// TIA Portal V21 export
FUNCTION_BLOCK "FB101"   // FB101, LAD
TITLE = FB101
{ S7_Optimized_Access := 'TRUE' }
AUTHOR : PRECISE
FAMILY : PRECISE
// TIMER (RETENTIVE)
// stored: AutoNumber false, MemoryReserve 100, SetENOAutomatically false
   VAR_INPUT
      Enable : Bool;
      Running : Bool;
      Reset : Bool;
      SecPulse : Bool;
      AlwaysTrue : Bool;
      TimeBaseSel : Bool;   // Time Base Selection: 0-second/1-minute
      TimeMin : Int;
      TimeSec : Int;
   END_VAR
   VAR_OUTPUT
      Done : Bool;
      TimeMinPV : DInt;
      TimeSecPV : DInt;
   END_VAR
   VAR_IN_OUT
      TimeSV : DInt;
      TimePV : DInt;
      TempBit : Bool;
   END_VAR
BEGIN

REGION Network 1: Set Time Min/Sec
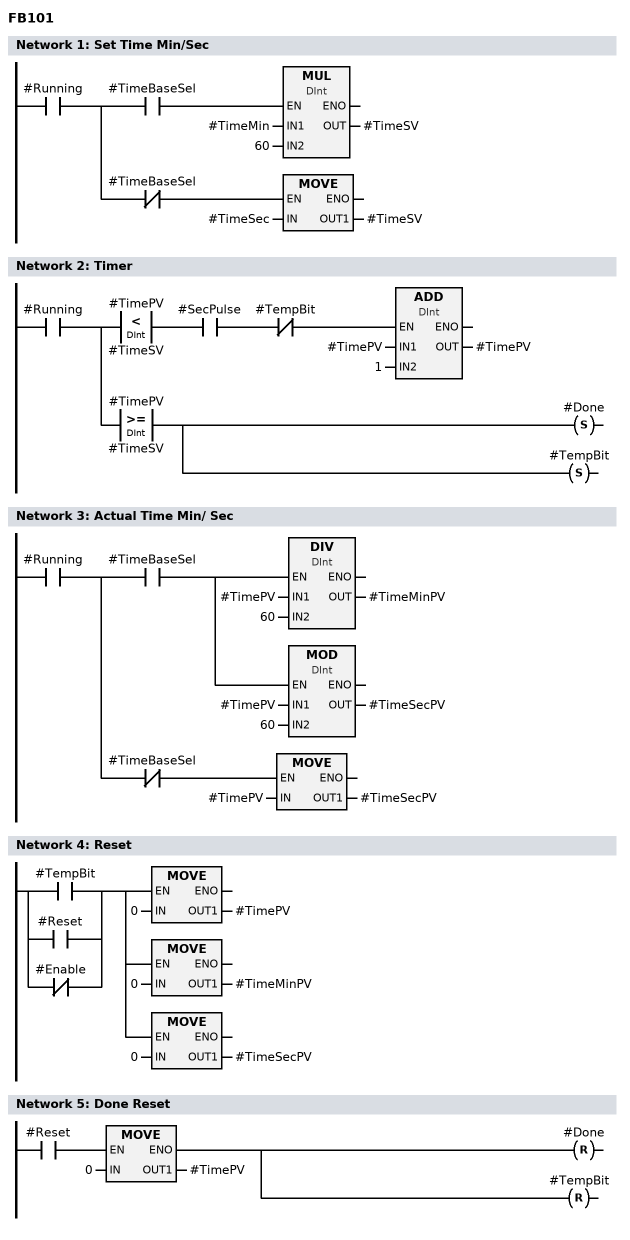
   RUNG wire#powerrail
      Contact( #Running )
      wire#w1
      Contact( #TimeBaseSel )
      { S7_Templates := "SrcType := DInt"; S7_GenerateENO := "TRUE" } Mul(in1 := #TimeMin, in2 := 60, out => #TimeSV)
   END_RUNG
   RUNG wire#w1
      I_Contact( #TimeBaseSel )
      { S7_GenerateENO := "TRUE" } Move(in := #TimeSec, out1 => #TimeSV)
   END_RUNG
   // the same network as SCL:
   IF #Running AND #TimeBaseSel THEN #TimeSV := #TimeMin * 60; END_IF;
   IF #Running AND NOT #TimeBaseSel THEN #TimeSV := #TimeSec; END_IF;
END_REGION

REGION Network 2: Timer
   RUNG wire#powerrail
      Contact( #Running )
      wire#w1
      { S7_Templates := "SrcType := DInt" } LT_Contact(in1 := #TimePV, in2 := #TimeSV)
      Contact( #SecPulse )
      I_Contact( #TempBit )
      { S7_Templates := "SrcType := DInt"; S7_GenerateENO := "TRUE" } Add(in1 := #TimePV, in2 := 1, out => #TimePV)
   END_RUNG
   RUNG wire#w1
      { S7_Templates := "SrcType := DInt" } GE_Contact(in1 := #TimePV, in2 := #TimeSV)
      wire#w2
      S_Coil( #Done )
   END_RUNG
   RUNG wire#w2
      S_Coil( #TempBit )
   END_RUNG
   // the same network as SCL:
   IF #Running AND (#TimePV < #TimeSV) AND #SecPulse AND NOT #TempBit THEN #TimePV := #TimePV + 1; END_IF;
   IF #Running AND (#TimePV >= #TimeSV) THEN
       #Done := TRUE;
       #TempBit := TRUE;
   END_IF;
END_REGION

REGION Network 3: Actual Time Min/ Sec
   RUNG wire#powerrail
      Contact( #Running )
      wire#w1
      Contact( #TimeBaseSel )
      wire#w2
      { S7_Templates := "SrcType := DInt"; S7_GenerateENO := "TRUE" } Div(in1 := #TimePV, in2 := 60, out => #TimeMinPV)
   END_RUNG
   RUNG wire#w2
      { S7_Templates := "SrcType := DInt"; S7_GenerateENO := "TRUE" } Mod(in1 := #TimePV, in2 := 60, out => #TimeSecPV)
   END_RUNG
   RUNG wire#w1
      I_Contact( #TimeBaseSel )
      { S7_GenerateENO := "TRUE" } Move(in := #TimePV, out1 => #TimeSecPV)
   END_RUNG
   // the same network as SCL:
   IF #Running AND #TimeBaseSel THEN
       #TimeMinPV := #TimePV / 60;
       #TimeSecPV := #TimePV MOD 60;
   END_IF;
   IF #Running AND NOT #TimeBaseSel THEN #TimeSecPV := #TimePV; END_IF;
END_REGION

REGION Network 4: Reset
   RUNG wire#powerrail
      Contact( #TempBit )
      wire#w1
      { S7_GenerateENO := "TRUE" } Move(in := 0, out1 => #TimePV)
   END_RUNG
   RUNG wire#powerrail
      Contact( #Reset )
   END_RUNG wire#w1
   RUNG wire#powerrail
      I_Contact( #Enable )
   END_RUNG wire#w1
   RUNG wire#w1
      { S7_GenerateENO := "TRUE" } Move(in := 0, out1 => #TimeMinPV)
   END_RUNG
   RUNG wire#w1
      { S7_GenerateENO := "TRUE" } Move(in := 0, out1 => #TimeSecPV)
   END_RUNG
   // the same network as SCL:
   IF #TempBit OR #Reset OR NOT #Enable THEN
       #TimePV := 0;
       #TimeMinPV := 0;
       #TimeSecPV := 0;
   END_IF;
END_REGION

REGION Network 5: Done Reset
   RUNG wire#powerrail
      Contact( #Reset )
      { S7_GenerateENO := "TRUE" } Move(in := 0, out1 => #TimePV)
      wire#w1
      R_Coil( #Done )
   END_RUNG
   RUNG wire#w1
      R_Coil( #TempBit )
   END_RUNG
   // the same network as SCL:
   // ENO of a box is taken as its EN; it also drops when the box reports an error
   IF #Reset THEN
       #TimePV := 0;
       #Done := FALSE;
       #TempBit := FALSE;
   END_IF;
END_REGION
END_FUNCTION_BLOCK
